// TIA Portal V19 export
FUNCTION_BLOCK "F_Zone00_FB"   // FB193, F_LAD
TITLE = SAFETY ZONE 00 - OUTSIDE SAFETY DOORS
// stored: Access Published
   VAR
      F_Sinamics_CoilCar : "FDevice_Sinamics_FB";
   END_VAR
   VAR CONSTANT
      COILCAR_S120_STOPPING_TIME : Time := t#2S;
   END_VAR
BEGIN

REGION Network 1: < < < < < < < < < < ZONE SAFETY INTERFACE > > > > > > > > > >
END_REGION

REGION Network 2: Cumulative Zone Safety
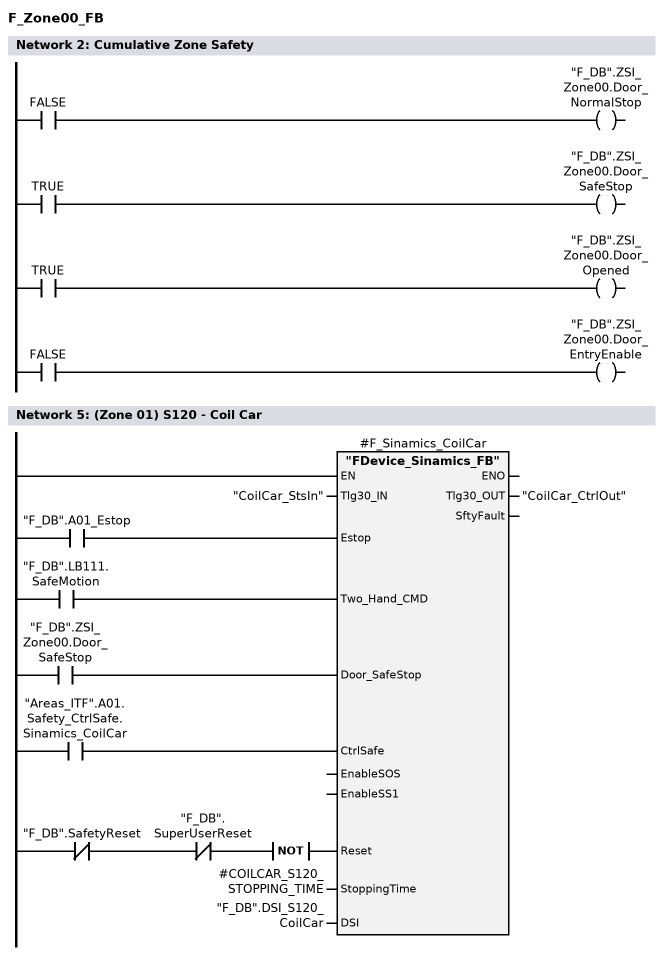
   RUNG wire#powerrail
      Contact( FALSE )
      Coil( "F_DB".ZSI_Zone00.Door_NormalStop )
   END_RUNG
   RUNG wire#powerrail
      Contact( TRUE )
      Coil( "F_DB".ZSI_Zone00.Door_SafeStop )
   END_RUNG
   RUNG wire#powerrail
      Contact( TRUE )
      Coil( "F_DB".ZSI_Zone00.Door_Opened )
   END_RUNG
   RUNG wire#powerrail
      Contact( FALSE )
      Coil( "F_DB".ZSI_Zone00.Door_EntryEnable )
   END_RUNG
   // the same network as SCL:
   "F_DB".ZSI_Zone00.Door_NormalStop := FALSE;
   "F_DB".ZSI_Zone00.Door_SafeStop := TRUE;
   "F_DB".ZSI_Zone00.Door_Opened := TRUE;
   "F_DB".ZSI_Zone00.Door_EntryEnable := FALSE;
END_REGION

REGION Network 3: < < < < < < < < < < DEVICES CONTACTORS > > > > > > > > > >
END_REGION

REGION Network 4: < < < < < < < < < < DEVICES S120 > > > > > > > > > >
END_REGION

REGION Network 5: (Zone 01) S120 - Coil Car
   RUNG wire#powerrail
      #F_Sinamics_CoilCar(Estop := wire#w1, Two_Hand_CMD := wire#w2, Door_SafeStop := wire#w3, CtrlSafe := wire#w4, Reset := wire#w5, Tlg30_IN := "CoilCar_StsIn", EnableSOS :=, EnableSS1 :=, StoppingTime := #COILCAR_S120_STOPPING_TIME, DSI := "F_DB".DSI_S120_CoilCar, Tlg30_OUT => "CoilCar_CtrlOut", SftyFault =>)
   END_RUNG
   RUNG wire#powerrail
      Contact( "F_DB".A01_Estop )
   END_RUNG wire#w1
   RUNG wire#powerrail
      Contact( "F_DB".LB111.SafeMotion )
   END_RUNG wire#w2
   RUNG wire#powerrail
      Contact( "F_DB".ZSI_Zone00.Door_SafeStop )
   END_RUNG wire#w3
   RUNG wire#powerrail
      Contact( "Areas_ITF".A01.Safety_CtrlSafe.Sinamics_CoilCar )
   END_RUNG wire#w4
   RUNG wire#powerrail
      I_Contact( "F_DB".SafetyReset )
      I_Contact( "F_DB".SuperUserReset )
      Not()
   END_RUNG wire#w5
   // the same network as SCL:
   #F_Sinamics_CoilCar(Tlg30_IN := "CoilCar_StsIn",   // "FDevice_Sinamics_FB"
                       Estop := "F_DB".A01_Estop,
                       Two_Hand_CMD := "F_DB".LB111.SafeMotion,
                       Door_SafeStop := "F_DB".ZSI_Zone00.Door_SafeStop,
                       CtrlSafe := "Areas_ITF".A01.Safety_CtrlSafe.Sinamics_CoilCar,
                       Reset := NOT (NOT "F_DB".SafetyReset AND NOT "F_DB".SuperUserReset),
                       StoppingTime := #COILCAR_S120_STOPPING_TIME,
                       DSI := "F_DB".DSI_S120_CoilCar,
                       Tlg30_OUT => "CoilCar_CtrlOut");
END_REGION
END_FUNCTION_BLOCK
